{attribute 'GeneratedUsingTerminal: EK1200-1b58-0000'}
{attribute addProperty BoxType "EK1200-1b58-0000"}
{attribute addProperty Description "EK1200-7000 EtherCAT Power supply (1,5A E-Bus)"}
{attribute addProperty Physics "YK"}
{attribute addProperty Id "EK1200"}
{attribute addProperty CRC "20777801"}
{attribute addProperty Size "0"}
TYPE EK1200_013D0B49 EXTENDS EtcSlaveBoxBase_77A0E4A7 :
STRUCT
END_STRUCT
END_TYPE

(* stored: Version 1.2.0.0, ProductVersion 3.1.4024.11
   DUT EK1200_013D0B49: Id {90b12bf1-29fc-431c-9268-fcca9401e79a} *)
